// TIA Portal V21 export
FUNCTION_BLOCK "BATCH LINE PRINT"   // FB5, LAD
{ S7_Optimized_Access := 'TRUE' }
// stored: MemoryReserve 100, SetENOAutomatically false
   VAR_INPUT
      PrintInetrval : Int;
      SecPulse : Bool;
   END_VAR
   VAR_IN_OUT
      ResetBatchTimer : Bool;
      BatchSelected : Bool;
   END_VAR
   VAR
      IEC_Counter_0_Instance { S7_SetPoint := 'True'} : CTU_INT;
   END_VAR
BEGIN

REGION Network 2
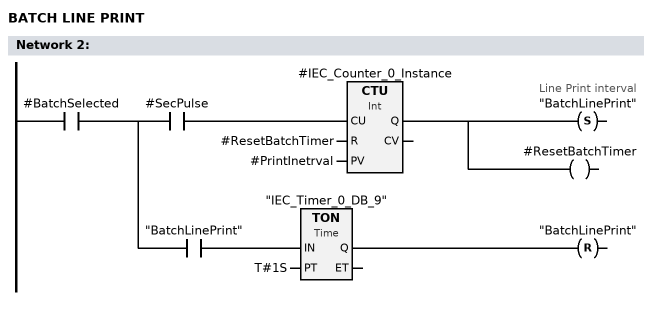
   RUNG wire#powerrail
      Contact( #BatchSelected )
      wire#w1
      Contact( #SecPulse )
      { S7_Templates := "value_type := Int" } #IEC_Counter_0_Instance.CTU(r := #ResetBatchTimer, pv := #PrintInetrval, cv =>)
      wire#w2
      S_Coil( "BatchLinePrint" )   // Line Print interval
   END_RUNG
   RUNG wire#w2
      Coil( #ResetBatchTimer )
   END_RUNG
   RUNG wire#w1
      Contact( "BatchLinePrint" )
      { S7_Templates := "time_type := Time" } "IEC_Timer_0_DB_9".TON(pt := T#1S, et =>)
      R_Coil( "BatchLinePrint" )
   END_RUNG
   // the same network as SCL:
   #IEC_Counter_0_Instance(CU := #BatchSelected AND #SecPulse, R := #ResetBatchTimer, PV := #PrintInetrval);   // CTU
   IF #IEC_Counter_0_Instance.Q THEN
       "BatchLinePrint" := TRUE;   // Line Print interval
   END_IF;
   #ResetBatchTimer := #IEC_Counter_0_Instance.Q;
   "IEC_Timer_0_DB_9".TON(IN := #BatchSelected AND "BatchLinePrint", PT := T#1S);
   IF "IEC_Timer_0_DB_9".Q THEN "BatchLinePrint" := FALSE; END_IF;
END_REGION
END_FUNCTION_BLOCK
